RoboDK station: fanuc_demo.rdk

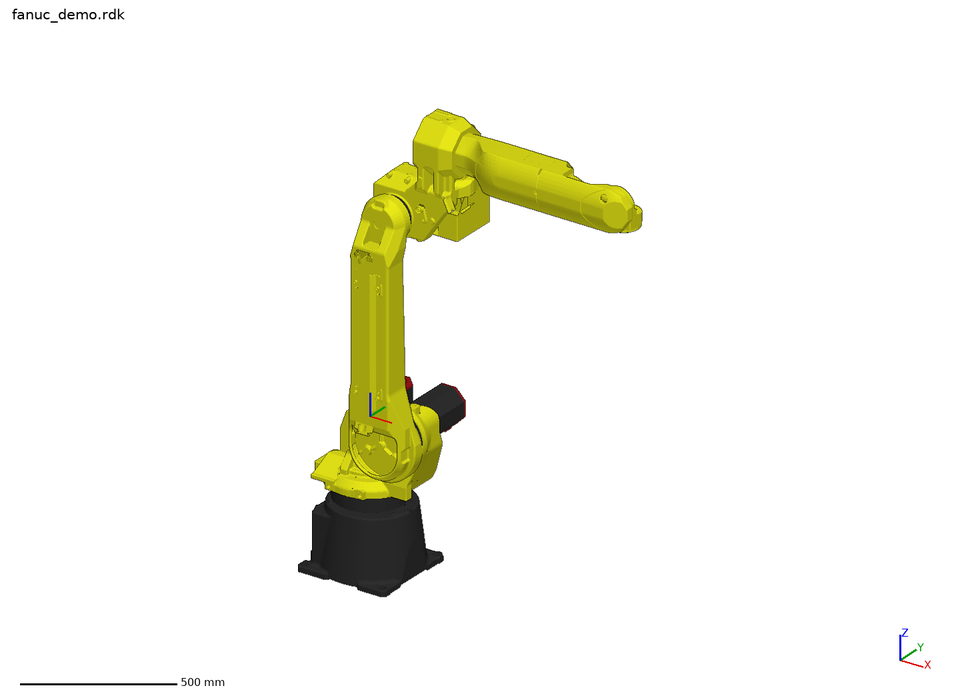
[picture v0: the station drawn from its stored meshes, robots at their saved joint values, targets as dots, program paths as lines]
Station fanuc_demo (saved by RoboDK 5.5.3). Poses are relative to the parent item; angles as X-Y-Z fixed-axis rotations.
Station parameters (name, value as stored): LIN64
  - frame Fanuc M-20iA Base at (0, 1000, 525) mm
    - robot Fanuc M-20iA: 6 axes, payload 20 kg, reach 1811 mm, repeatability 0.08 mm, weight 250 kg
        modified DH rows (alpha deg, a mm, theta deg, d mm): 0, 0, 0, 525; -90, 150, -90, 0; 0, 790, 0, 0; -90, 250, 0, 835; 90, 0, 0, 0; -90, 0, 0, 100
        base shift (0, 0, -525) mm
        joint limits [-185, -110, -75, -200, -180, -450] to [185, 110, 245, 200, 180, 450]; home [0, 0, 0, 0, 0, 0]; saved at [0, 0, 0, 0, -90, 0]
  - Python program Demo1 (listed below)
  - Python program reset (listed below)

--- Python program Demo1 ---
# Type help("robodk.robolink") or help("robodk.robomath") for more information
# Press F5 to run the script
# Documentation: https://robodk.com/doc/en/RoboDK-API.html
# Reference:     https://robodk.com/doc/en/PythonAPI/robodk.html
# Note: It is not required to keep a copy of this file, your Python script is saved with your RDK project

from robodk.robolink import *  # API to communicate with RoboDK
from robodk.robomath import *  # basic matrix operations
# Link to RoboDK
# RDK = Robolink()
RDK = Robolink()

# Notify user:
print('To edit this program:\nright click on the Python program, then, select "Edit Python script"')

# Program example:
item = RDK.Item('base')
if item.Valid():
    print('Item selected: ' + item.Name())
    print('Item posistion: ' + repr(item.Pose()))

print('Items in the station:')
itemlist = RDK.ItemList()
robot = RDK.ItemUserPick('Select a robot', ITEM_TYPE_ROBOT)
print(itemlist)

robot.MoveJ([0.000, 37, 0.000, -0.000, -90.000, -0.000])

--- Python program reset ---
# Type help("robodk.robolink") or help("robodk.robomath") for more information
# Press F5 to run the script
# Documentation: https://robodk.com/doc/en/RoboDK-API.html
# Reference:     https://robodk.com/doc/en/PythonAPI/robodk.html
# Note: It is not required to keep a copy of this file, your Python script is saved with your RDK project

from robodk.robolink import *  # API to communicate with RoboDK
from robodk.robomath import *  # basic matrix operations
# Link to RoboDK
# RDK = Robolink()
RDK = Robolink()

# Notify user:
print('To edit this program:\nright click on the Python program, then, select "Edit Python script"')

# Program example:
item = RDK.Item('base')
if item.Valid():
    print('Item selected: ' + item.Name())
    print('Item posistion: ' + repr(item.Pose()))

print('Items in the station:')
itemlist = RDK.ItemList()
robot = RDK.ItemUserPick('Select a robot', ITEM_TYPE_ROBOT)
print(itemlist)

robot.MoveJ([0.000, 0.000, 0.000, -0.000, -90.000, -0.000])
